FUNCTION_BLOCK Test_F_UDINT_TO_DINT_Conversion EXTENDS TUnitTestBase
VAR
    InputValue : UDINT;
    ConvertedValue : DINT;
END_VAR

InputValue := 2147483648; // too big
ConvertedValue := F_UDINT_TO_DINT(InputValue); // limit to largest DINT

Assertion.AssertEquals_DINT(
    Expected:= 2147483647, 
    Actual:= ConvertedValue, 
    VariableName:= 'ConvertedValue');
    
TestFinished();

END_FUNCTION_BLOCK

(* stored: Version 1.1.0.1, ProductVersion 3.1.4024.4
   POU Test_F_UDINT_TO_DINT_Conversion: Id {95f19bb1-69bf-4f94-a858-73cae353435d}, SpecialFunc None *)
